TYPE ST_CommandsATS :
STRUCT
	ToGen				: BOOL := FALSE;
	ToLine				: BOOL := FALSE;
	OFF					: BOOL := FALSE;
END_STRUCT
END_TYPE

(* stored: Version 1.1.0.1, ProductVersion 3.1.4026.18
   DUT ST_CommandsATS: Id {c476504c-3b4e-41ba-bf30-a5a2670a966a} *)
